TYPE WriteXmlProcessArgs :
STRUCT
	///Full path of the filename to write
	filePath: STRING;
END_STRUCT
END_TYPE

(* stored: Version 1.1.0.1, ProductVersion 3.1.4019.2
   DUT WriteXmlProcessArgs: Id {63ab46cd-6cfd-4d39-b332-a74afa08e063} *)
